FUNCTION_BLOCK RotatingArmReset (* Composite Function Block Type *)
  (* Standard: 61499-2 *)
  (* Version 0.0, 2/11/2018, Sandeep Patil, nxtControl GmbH, template *)
  PACKAGE Main;
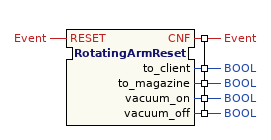
  EVENT_INPUT
    RESET; (* Initialization Request *)
  END_EVENT
  EVENT_OUTPUT
    CNF WITH to_client, to_magazine, vacuum_on, vacuum_off; (* Execution Confirmation *)
  END_EVENT
  VAR_OUTPUT
    to_client : BOOL;
    to_magazine : BOOL;
    vacuum_on : BOOL;
    vacuum_off : BOOL;
  END_VAR
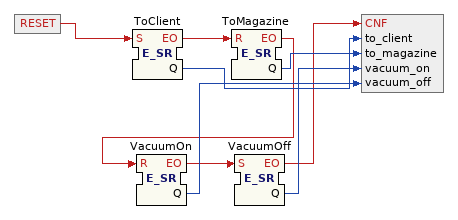
  FBS
    ToClient : E_SR;
    ToMagazine : E_SR;
    VacuumOff : E_SR;
    VacuumOn : E_SR;
  END_FBS
  EVENT_CONNECTIONS
    RESET TO ToClient.S;
    ToClient.EO TO ToMagazine.R;
    VacuumOff.EO TO CNF;
    ToMagazine.EO TO VacuumOn.R;
    VacuumOn.EO TO VacuumOff.S;
  END_CONNECTIONS
  DATA_CONNECTIONS
    ToClient.Q TO to_client;
    ToMagazine.Q TO to_magazine;
    VacuumOff.Q TO vacuum_on;
    VacuumOn.Q TO vacuum_off;
  END_CONNECTIONS
END_FUNCTION_BLOCK
